Staubli VAL3: F3_delete.pgx

program F3_delete()
  local num l_ni
begin
  //delete points
  //  nTotalPoints=size(pfrmCad)
  //  if nTotalPoints>1
  //    //      for l_ni=nTotalPoints to 2 step -1
  //    //        $ddel(pfrmCad,l_ni-1)
  //    ////        nTotalPoints=nTotalPoints-1
  //    ////        nScrPts=nTotalPoints
  //    //
  //    //      endFor
  //    //       call hmi_refreshmain()
  //    for l_ni=nTotalPoints to 2 step -1
  //      $ddel(pfrmCad,nTotalPoints-1)
  //      nTotalPoints=nTotalPoints-1
  //      nScrPts=nTotalPoints
  //    endFor
  //    call hmi_refreshmain()
  //  else
  //    popUpMsg("No points existed")
  //  endIf
end
